FUNCTION_BLOCK FB_Fast_brake
VAR_INPUT
	Lh_depth:REAL;
	Rh_depth:REAL;
	Speed:REAL;
	Fast_brake_top_depth:REAL;
	Fast_brake_bottom_depth:REAL;
	Fast_brake_speed:REAL;
	Speed_hysteresis:REAL;
	Off_delay_after_brakes_on:TIME;
	Check_speed:REAL;
END_VAR
VAR_OUTPUT
	Valve:BOOL;
	Active_above_check_speed:BOOL;
END_VAR
VAR
	FB_CTRL_HYSTERESIS_0: FB_CTRL_HYSTERESIS;
	TON_0: TON;
END_VAR

M_Fast_brake();

METHOD M_Fast_brake
VAR_INPUT
END_VAR
{warning "TODO: HYSTERESIS block needs to be figured out and made to work correctly."}
VAR_INST // added by the converter: edge detectors and wires of the graphical bodies
    _w1, _w2, _w3, _w4, _w5, _w7 : BOOL;
    _w6 : ANY;
END_VAR
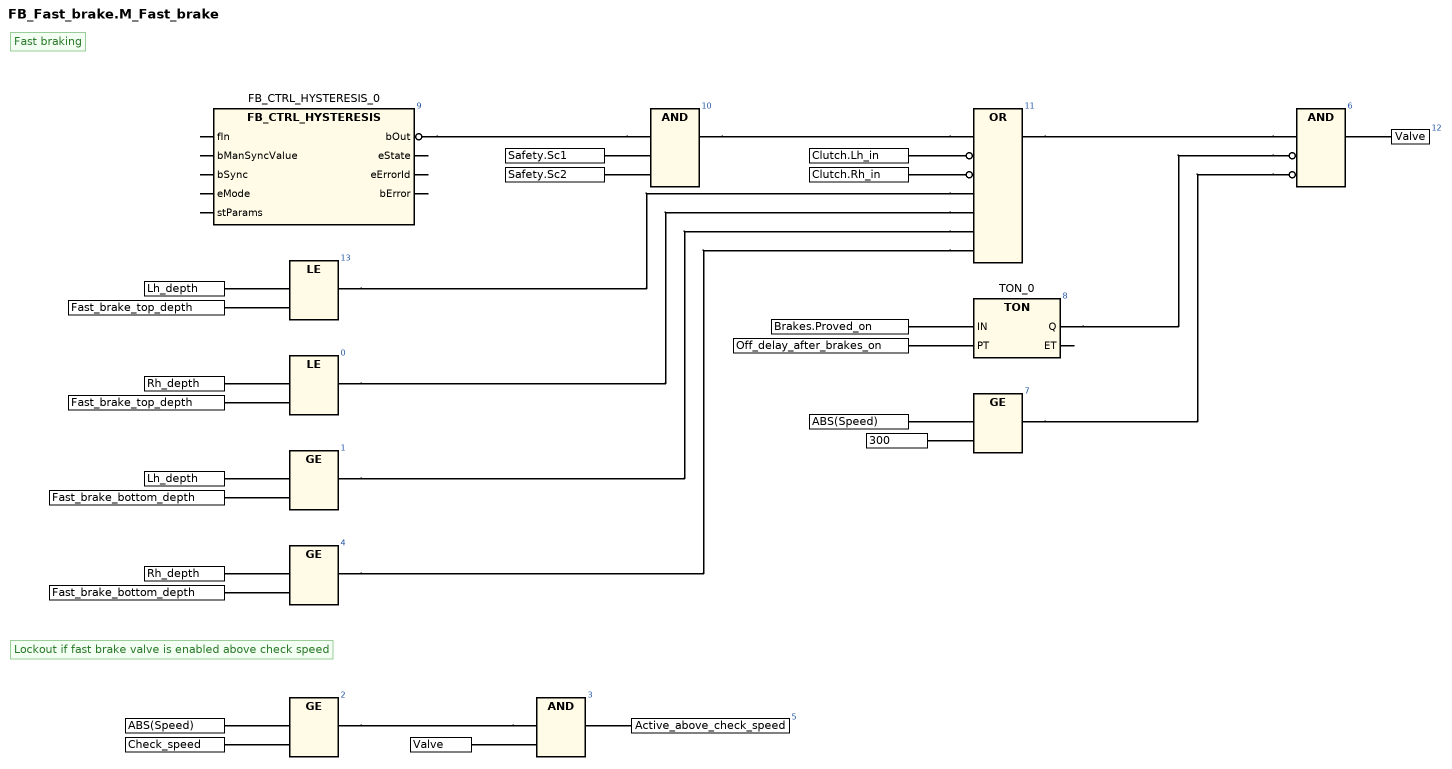
_w1 := Rh_depth <= Fast_brake_top_depth;
_w2 := Lh_depth >= Fast_brake_bottom_depth;
// Lockout if fast brake valve is enabled above check speed
_w3 := Rh_depth >= Fast_brake_bottom_depth;
Active_above_check_speed := (ABS(Speed)) >= Check_speed AND Valve;
_w6 := _w4 AND NOT TON_0.Q AND NOT _w5;
_w5 := (ABS(Speed)) >= 300;
TON_0(IN := Brakes.Proved_on, PT := Off_delay_after_brakes_on); // TON
// Fast braking
FB_CTRL_HYSTERESIS_0(); // FB_CTRL_HYSTERESIS
_w4 := NOT FB_CTRL_HYSTERESIS_0.bOut AND Safety.Sc1 AND Safety.Sc2 OR NOT Clutch.Lh_in OR NOT Clutch.Rh_in OR _w7 OR _w1 OR _w2 OR _w3;
Valve := _w6;
_w7 := Lh_depth <= Fast_brake_top_depth;
END_METHOD

END_FUNCTION_BLOCK

(* stored: Version 1.1.0.1, ProductVersion 3.1.4024.0
   POU FB_Fast_brake: Id {2eeb86e2-90f8-4305-92b6-a1d1d64111a9}, SpecialFunc None
   Method M_Fast_brake: Id {e8069fff-640c-44da-9149-5c9af6ec7085} *)
